{attribute addProperty BoxType "AT2041-0250-0020"}
{attribute addProperty Id "A_0102_AT2041_5250_0019_AT2041_5250AT2041_3DCFC8D064080"}
{attribute addProperty CRC "271374235"}
{attribute addProperty SizeInBites "640"}
{attribute addProperty SizeInBytes "80"}
TYPE A_0042_AT2041_0250_0020_102CD79B EXTENDS AT2041_9506A482 :
STRUCT
	{attribute addProperty Name "A_0102_AT2041_5250_0019_AT2041_5250"}
	A_0102_AT2041_5250_0019_AT2041_5250 : AT2041_3DCFC8D0;
END_STRUCT
END_TYPE

(* stored: Version 1.2.0.0, ProductVersion 3.1.4024.9
   DUT A_0042_AT2041_0250_0020_102CD79B: Id {072f1c1c-6ac5-4c33-87e9-1e167405a7ec} *)
